(* IEC 61131-3 sources: RL_MAR/experiments/comparison/autoplc/results/gpt-4o-mini_20260511_164212/med_89, 1 file *)

(* ---- med_89_1.st ---- *)
FUNCTION_BLOCK SoilTestingDeviceControl
VAR_INPUT
    StartButton : BOOL; (* Input for starting the testing process *)
    SoilSampleDetected : BOOL; (* Input for detecting soil sample *)
END_VAR

VAR_OUTPUT
    NutrientPump : BOOL; (* Output to control nutrient pump *)
    pHAdjustmentPump : BOOL; (* Output to control pH adjustment pump *)
END_VAR

VAR
    pHSensorValue : REAL; (* Simulated pH sensor value *)
    NutrientSensorValue : REAL; (* Simulated nutrient sensor value *)
    TestingStatus : INT; (* Status: 0=Idle, 1=Testing, 2=Completed *)
    NutrientThreshold : REAL := 0.7; (* Nutrient level threshold for analysis *)
    pHThreshold : REAL := 6.5; (* pH level threshold for analysis *)
END_VAR

(* Main control logic *)
IF TestingStatus = 0 THEN
    (* Initialization *)
    pHSensorValue := 7.0;
    NutrientSensorValue := 0.5;
END_IF;

IF StartButton AND TestingStatus = 0 THEN
    (* Start Testing *)
    TestingStatus := 1; (* Transition to Testing state *)
    NutrientPump := TRUE; (* Activate Nutrient Pump *)
    pHAdjustmentPump := TRUE; (* Activate pH Adjustment Pump *)
END_IF;

IF TestingStatus = 1 THEN
    (* During Testing *)
    IF SoilSampleDetected THEN
        (* Check conditions for completion *)
        IF NutrientSensorValue >= NutrientThreshold AND pHSensorValue <= pHThreshold THEN
            TestingStatus := 2; (* Transition to Completed state *)
            NutrientPump := FALSE; (* Deactivate Nutrient Pump *)
            pHAdjustmentPump := FALSE; (* Deactivate pH Adjustment Pump *)
        END_IF;
    END_IF;

    (* Simulated Sensor Value Updates *)
    IF NutrientSensorValue < 0.9 THEN
        NutrientSensorValue := NutrientSensorValue + 0.1; (* Increment Nutrient Sensor Value *)
    END_IF;

    IF pHSensorValue > 4.0 THEN
        pHSensorValue := pHSensorValue - 0.5; (* Decrement pH Sensor Value *)
    END_IF;
END_IF;

END_FUNCTION_BLOCK
